DATA_BLOCK "DB2015_M"
TITLE = DB2015_M
{ S7_Optimized_Access := 'FALSE' }
AUTHOR : ABH
FAMILY : ZeusControl
VERSION : 1.0
//Bloque de datos motor.
   STRUCT
      M { S7_SetPoint := 'False'} : Array[0.."N_MAX_DISP_M"] of "UDT_ZC_DISP_M";
      Mux { S7_SetPoint := 'False'} : Array[0.."N_MAX_MUX_DISP"] of "UDT_ZC_DISP_MUX_M";
      Agrup : Array[0.."N_MAX_DISP_AGRUP"] of "UDT_ZC_DISP_AGRUP";
   END_STRUCT;


BEGIN
   M[0].Hmi_Estado := 0;
   M[0].Estado_AutoMan := FALSE;
   M[0].Estado_Activado := FALSE;
   M[0].Estado_Enclavado := FALSE;
   M[0].Estado_EntradaTermico := FALSE;
   M[0].Estado_EntradaConfMarcha := FALSE;
   M[0].Alarmas_Termico := FALSE;
   M[0].Alarmas_ConfirmacionMarcha := FALSE;
   M[0].Alarmas_Mantenimiento := FALSE;
   M[0].Alarmas_General := FALSE;
   M[0].Orden_ActivarManual := FALSE;
   M[0].Orden_ActivarAuto := FALSE;
   M[0].Orden_ResetHoras := FALSE;
   M[0].Config_Habilitar := FALSE;
   M[0].Config_HabilitarRetornoTermico := TRUE;
   M[0].Config_HabilitarInvertirTermico := FALSE;
   M[0].Config_HabilitarRetornoConfMarcha := TRUE;
   M[0].Config_HabilitarInvertirConfMarcha := FALSE;
   M[0].Config_HabilitarMantenimiento := FALSE;
   M[0].Aux_oldActivado := FALSE;
   M[0].Aux_oldAlarma := FALSE;
   M[0].Aux_oldAutoMan := FALSE;
   M[0].Estado_SeguridadOk := TRUE;
   M[0].Config_GrupoAlarma := 0;
   M[0].Config_DireccionSalidaByte := 0;
   M[0].Config_DireccionSalidaBit := 0;
   M[0].Config_DireccionRetTermicoByte := 0;
   M[0].Config_DireccionRetTermicoBit := 0;
   M[0].Config_DireccionRetConfMarchaByte := 0;
   M[0].Config_DireccionRetConfMarchaBit := 0;
   M[0].Tiempos_SetPointTiempoAlarma := 10;
   M[0].Tiempos_Alarma := 0;
   M[0].Tiempos_SetPointMantenimiento := 2000.0;
   M[0].Tiempos_Mantenimiento := 0.0;
   M[1].Hmi_Estado := 1;
   M[1].Estado_AutoMan := FALSE;
   M[1].Estado_Activado := FALSE;
   M[1].Estado_Enclavado := FALSE;
   M[1].Estado_EntradaTermico := FALSE;
   M[1].Estado_EntradaConfMarcha := FALSE;
   M[1].Alarmas_Termico := FALSE;
   M[1].Alarmas_ConfirmacionMarcha := FALSE;
   M[1].Alarmas_Mantenimiento := FALSE;
   M[1].Alarmas_General := FALSE;
   M[1].Orden_ActivarManual := FALSE;
   M[1].Orden_ActivarAuto := FALSE;
   M[1].Orden_ResetHoras := FALSE;
   M[1].Config_Habilitar := TRUE;
   M[1].Config_HabilitarRetornoTermico := FALSE;
   M[1].Config_HabilitarInvertirTermico := FALSE;
   M[1].Config_HabilitarRetornoConfMarcha := TRUE;
   M[1].Config_HabilitarInvertirConfMarcha := FALSE;
   M[1].Config_HabilitarMantenimiento := FALSE;
   M[1].Aux_oldActivado := FALSE;
   M[1].Aux_oldAlarma := FALSE;
   M[1].Aux_oldAutoMan := FALSE;
   M[1].Estado_SeguridadOk := TRUE;
   M[1].Config_GrupoAlarma := 0;
   M[1].Config_DireccionSalidaByte := 100;
   M[1].Config_DireccionSalidaBit := 3;
   M[1].Config_DireccionRetTermicoByte := 0;
   M[1].Config_DireccionRetTermicoBit := 0;
   M[1].Config_DireccionRetConfMarchaByte := 100;
   M[1].Config_DireccionRetConfMarchaBit := 6;
   M[1].Tiempos_SetPointTiempoAlarma := 10;
   M[1].Tiempos_Alarma := 0;
   M[1].Tiempos_SetPointMantenimiento := 2000.0;
   M[1].Tiempos_Mantenimiento := 4.633314;
   Mux[0].Habilitar := TRUE;
   Mux[0].ExisteCambio := FALSE;
   Mux[0].MaxVisible := FALSE;
   Mux[0].Index := 43;
   Mux[0].oldIndex := 43;
   Mux[0].M.Hmi_Estado := 1;
   Mux[0].M.Estado_AutoMan := FALSE;
   Mux[0].M.Estado_Activado := FALSE;
   Mux[0].M.Estado_Enclavado := FALSE;
   Mux[0].M.Estado_EntradaTermico := FALSE;
   Mux[0].M.Estado_EntradaConfMarcha := FALSE;
   Mux[0].M.Alarmas_Termico := FALSE;
   Mux[0].M.Alarmas_ConfirmacionMarcha := FALSE;
   Mux[0].M.Alarmas_Mantenimiento := FALSE;
   Mux[0].M.Alarmas_General := FALSE;
   Mux[0].M.Orden_ActivarManual := FALSE;
   Mux[0].M.Orden_ActivarAuto := FALSE;
   Mux[0].M.Orden_ResetHoras := FALSE;
   Mux[0].M.Config_Habilitar := TRUE;
   Mux[0].M.Config_HabilitarRetornoTermico := FALSE;
   Mux[0].M.Config_HabilitarInvertirTermico := FALSE;
   Mux[0].M.Config_HabilitarRetornoConfMarcha := TRUE;
   Mux[0].M.Config_HabilitarInvertirConfMarcha := FALSE;
   Mux[0].M.Config_HabilitarMantenimiento := FALSE;
   Mux[0].M.Aux_oldActivado := FALSE;
   Mux[0].M.Aux_oldAlarma := FALSE;
   Mux[0].M.Aux_oldAutoMan := FALSE;
   Mux[0].M.Estado_SeguridadOk := TRUE;
   Mux[0].M.Config_GrupoAlarma := 4;
   Mux[0].M.Config_DireccionSalidaByte := 501;
   Mux[0].M.Config_DireccionSalidaBit := 0;
   Mux[0].M.Config_DireccionRetTermicoByte := 0;
   Mux[0].M.Config_DireccionRetTermicoBit := 0;
   Mux[0].M.Config_DireccionRetConfMarchaByte := 501;
   Mux[0].M.Config_DireccionRetConfMarchaBit := 5;
   Mux[0].M.Tiempos_SetPointTiempoAlarma := 10;
   Mux[0].M.Tiempos_Alarma := 0;
   Mux[0].M.Tiempos_SetPointMantenimiento := 2000.0;
   Mux[0].M.Tiempos_Mantenimiento := 18.71946;
   Mux[1].Habilitar := TRUE;
   Mux[1].ExisteCambio := FALSE;
   Mux[1].MaxVisible := FALSE;
   Mux[1].Index := 0;
   Mux[1].oldIndex := 0;
   Mux[1].M.Hmi_Estado := 0;
   Mux[1].M.Estado_AutoMan := FALSE;
   Mux[1].M.Estado_Activado := FALSE;
   Mux[1].M.Estado_Enclavado := FALSE;
   Mux[1].M.Estado_EntradaTermico := FALSE;
   Mux[1].M.Estado_EntradaConfMarcha := FALSE;
   Mux[1].M.Alarmas_Termico := FALSE;
   Mux[1].M.Alarmas_ConfirmacionMarcha := FALSE;
   Mux[1].M.Alarmas_Mantenimiento := FALSE;
   Mux[1].M.Alarmas_General := FALSE;
   Mux[1].M.Orden_ActivarManual := FALSE;
   Mux[1].M.Orden_ActivarAuto := FALSE;
   Mux[1].M.Orden_ResetHoras := FALSE;
   Mux[1].M.Config_Habilitar := FALSE;
   Mux[1].M.Config_HabilitarRetornoTermico := TRUE;
   Mux[1].M.Config_HabilitarInvertirTermico := FALSE;
   Mux[1].M.Config_HabilitarRetornoConfMarcha := TRUE;
   Mux[1].M.Config_HabilitarInvertirConfMarcha := FALSE;
   Mux[1].M.Config_HabilitarMantenimiento := FALSE;
   Mux[1].M.Aux_oldActivado := FALSE;
   Mux[1].M.Aux_oldAlarma := FALSE;
   Mux[1].M.Aux_oldAutoMan := FALSE;
   Mux[1].M.Estado_SeguridadOk := TRUE;
   Mux[1].M.Config_GrupoAlarma := 0;
   Mux[1].M.Config_DireccionSalidaByte := 0;
   Mux[1].M.Config_DireccionSalidaBit := 0;
   Mux[1].M.Config_DireccionRetTermicoByte := 0;
   Mux[1].M.Config_DireccionRetTermicoBit := 0;
   Mux[1].M.Config_DireccionRetConfMarchaByte := 0;
   Mux[1].M.Config_DireccionRetConfMarchaBit := 0;
   Mux[1].M.Tiempos_SetPointTiempoAlarma := 10;
   Mux[1].M.Tiempos_Alarma := 0;
   Mux[1].M.Tiempos_SetPointMantenimiento := 2000.0;
   Mux[1].M.Tiempos_Mantenimiento := 0.0;
   Agrup[0].AlgunaEnManual := FALSE;
   Agrup[0].AlgunaAlarma := FALSE;
   Agrup[0].NuevaAlarma := FALSE;
   Agrup[1].AlgunaEnManual := FALSE;
   Agrup[1].AlgunaAlarma := FALSE;
   Agrup[1].NuevaAlarma := FALSE;

END_DATA_BLOCK

